FUNCTION_BLOCK PlottingStateMachine (* Template for a simple Basic Function Block Type *)
  (* Standard: 61499-2 *)
  (* Version 1.0, 2019-12-17, Mario *)
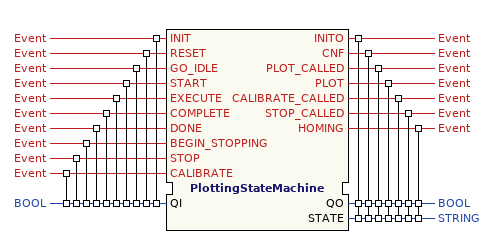
  EVENT_INPUT
    INIT WITH QI; (* Initialization Request *)
    RESET WITH QI; (* Reset plotter *)
    GO_IDLE WITH QI; (* Go into idle state *)
    START WITH QI; (* Initiate plotting *)
    EXECUTE WITH QI; (* Plot from file *)
    COMPLETE WITH QI; (* Finish plotting *)
    DONE WITH QI; (* Plotting complete *)
    BEGIN_STOPPING WITH QI; (* Get ready to go into stop state *)
    STOP WITH QI; (* Stop plotter *)
    CALIBRATE WITH QI; (* Go into calibrating mode *)
  END_EVENT
  EVENT_OUTPUT
    INITO WITH QO, STATE; (* Initialization Confirm *)
    CNF WITH QO, STATE; (* Execution Confirmation *)
    PLOT_CALLED WITH QO, STATE; (* Event to start plotting *)
    PLOT WITH STATE, QO; (* Start plotting *)
    CALIBRATE_CALLED WITH QO, STATE; (* Event to go into calibration mode *)
    STOP_CALLED WITH QO, STATE; (* Prepare to go into stop state *)
    HOMING WITH QO, STATE; (* Reset Plotter position to origin *)
  END_EVENT
  VAR_INPUT
    QI : BOOL; (* Input event qualifier *)
  END_VAR
  VAR_OUTPUT
    QO : BOOL; (* Output event qualifier *)
    STATE : STRING; (* Plotter State as String *)
  END_VAR
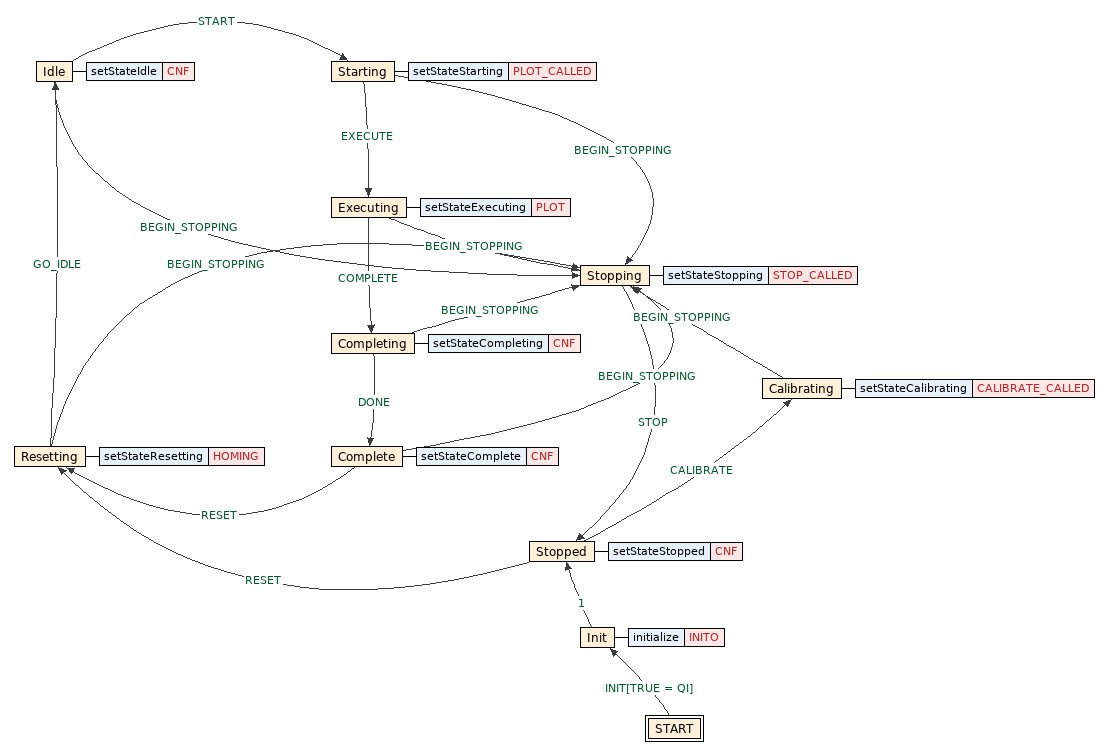
  EC_STATES
    START; (* Initial State *)
    Init : initialize -> INITO; (* Initialization *)
    Idle : setStateIdle -> CNF;
    Starting : setStateStarting -> PLOT_CALLED;
    Executing : setStateExecuting -> PLOT;
    Completing : setStateCompleting -> CNF;
    Complete : setStateComplete -> CNF;
    Resetting : setStateResetting -> HOMING;
    Stopping : setStateStopping -> STOP_CALLED;
    Stopped : setStateStopped -> CNF;
    Calibrating : setStateCalibrating -> CALIBRATE_CALLED;
  END_STATES
  EC_TRANSITIONS
    START TO Init := INIT[TRUE = QI];
    Init TO Stopped := 1;
    Stopped TO Calibrating := CALIBRATE;
    Stopping TO Stopped := STOP;
    Resetting TO Idle := GO_IDLE;
    Idle TO Starting := START;
    Starting TO Executing := EXECUTE;
    Executing TO Completing := COMPLETE;
    Completing TO Complete := DONE;
    Complete TO Resetting := RESET;
    Stopped TO Resetting := RESET;
    Calibrating TO Stopping := BEGIN_STOPPING;
    Executing TO Stopping := BEGIN_STOPPING;
    Completing TO Stopping := BEGIN_STOPPING;
    Complete TO Stopping := BEGIN_STOPPING;
    Resetting TO Stopping := BEGIN_STOPPING;
    Idle TO Stopping := BEGIN_STOPPING;
    Starting TO Stopping := BEGIN_STOPPING;
  END_TRANSITIONS
  ALGORITHM initialize IN ST: (* Initialization algorithm *)
QO := QI;
STATE := "NOT_INITIALIZED";
  END_ALGORITHM
  ALGORITHM deInitialize IN ST: (* Normally executed algorithm *)
QO := FALSE;
  END_ALGORITHM
  ALGORITHM normalOperation IN ST: (* new algorithm *)
QO := QI;

IF TRUE  = QI THEN
  (*  only perform normal operation of QI is true*)

END_IF;
  END_ALGORITHM
  ALGORITHM setStateResetting IN ST: (* new algorithm *)
STATE := "RESET";
  END_ALGORITHM
  ALGORITHM setStateIdle IN ST: (* new algorithm *)
STATE := "IDLE";
  END_ALGORITHM
  ALGORITHM setStateStarting IN ST: (* new algorithm *)
STATE := "STARTING";
  END_ALGORITHM
  ALGORITHM setStateExecuting IN ST: (* new algorithm *)
STATE := "EXECUTING";
  END_ALGORITHM
  ALGORITHM setStateCompleting IN ST: (* new algorithm *)
STATE := "COMPLETING";
  END_ALGORITHM
  ALGORITHM setStateComplete IN ST: (* new algorithm *)
STATE := "COMPLETE";
  END_ALGORITHM
  ALGORITHM setStateStopping IN ST: (* new algorithm *)
STATE := "STOPPING";
  END_ALGORITHM
  ALGORITHM setStateStopped IN ST: (* new algorithm *)
STATE := "STOPPED";
  END_ALGORITHM
  ALGORITHM setStateCalibrating IN ST: (* new algorithm *)
STATE := "CALIBRATING";
  END_ALGORITHM
END_FUNCTION_BLOCK
